PROGRAM analogSignals_ex06
VAR
	valvecontrol			: REAL;
	valveopening			: REAL;
	
	LIN_TRAFO 			: FB_Scale;
END_VAR

LIN_TRAFO(
	fIN:= valvecontrol, 
	fIN_min:= 0, 
	fIN_max:= 100, 
	fOUT_min:= 0, 
	fOUT_max:= 10, 
	fOUT=> valveopening);

END_PROGRAM

(* stored: Version 1.1.0.1
   POU analogSignals_ex06: Id {7821f3af-0438-4c5c-ae29-a4b263456196}, SpecialFunc None *)
